// Mitsubishi GX Works2 project: 1111   PLC: Q00J
// 1111111

PROGRAM MAIN
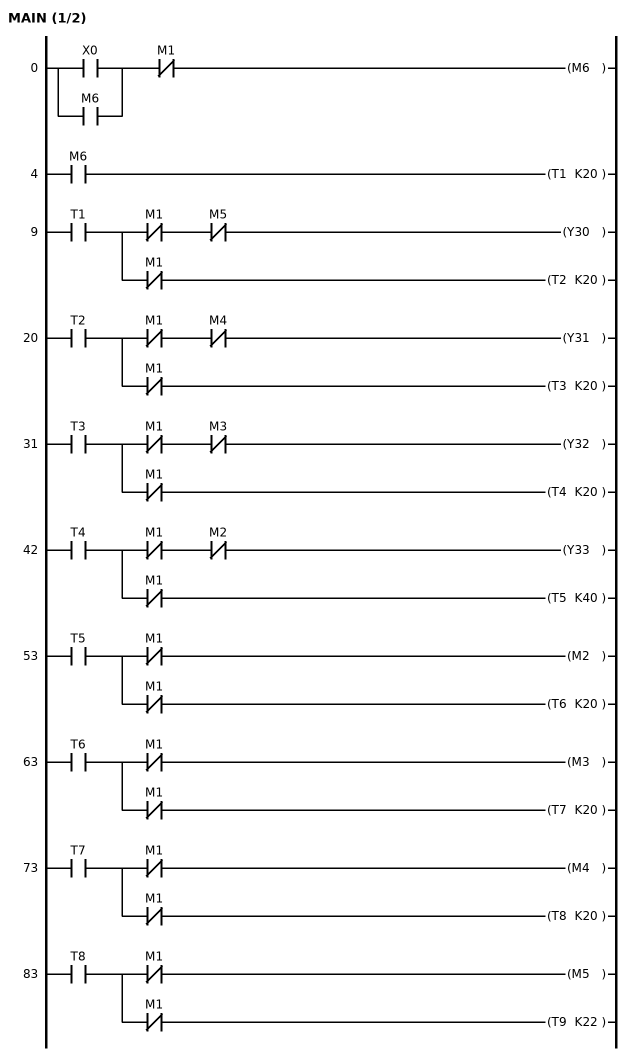
0     LD      X0
      OR      M6
      ANI     M1
      OUT     M6
4     LD      M6
      OUT     T1 K20
9     LD      T1
      MPS
      ANI     M1
      ANI     M5
      OUT     Y30
      MPP
      ANI     M1
      OUT     T2 K20
20    LD      T2
      MPS
      ANI     M1
      ANI     M4
      OUT     Y31
      MPP
      ANI     M1
      OUT     T3 K20
31    LD      T3
      MPS
      ANI     M1
      ANI     M3
      OUT     Y32
      MPP
      ANI     M1
      OUT     T4 K20
42    LD      T4
      MPS
      ANI     M1
      ANI     M2
      OUT     Y33
      MPP
      ANI     M1
      OUT     T5 K40
53    LD      T5
      MPS
      ANI     M1
      OUT     M2
      MPP
      ANI     M1
      OUT     T6 K20
63    LD      T6
      MPS
      ANI     M1
      OUT     M3
      MPP
      ANI     M1
      OUT     T7 K20
73    LD      T7
      MPS
      ANI     M1
      OUT     M4
      MPP
      ANI     M1
      OUT     T8 K20
83    LD      T8
      MPS
      ANI     M1
      OUT     M5
      MPP
      ANI     M1
      OUT     T9 K22
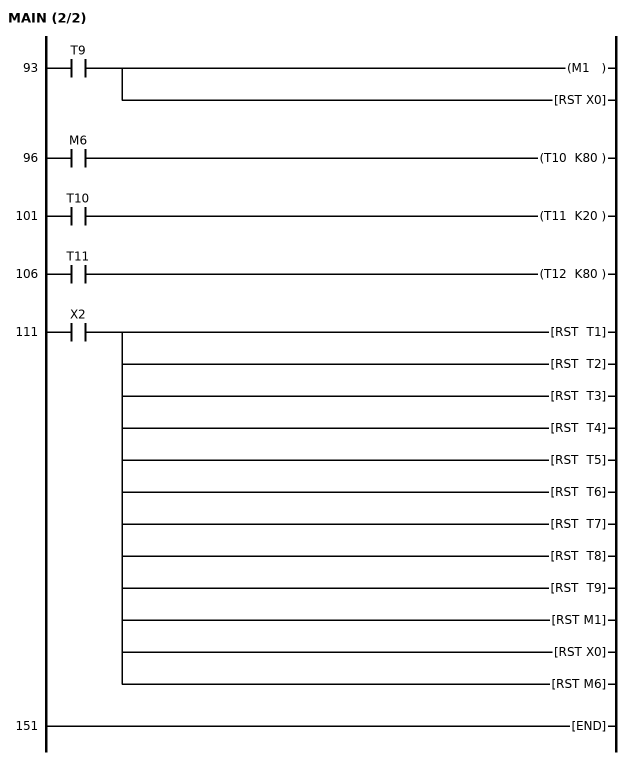
93    LD      T9
      OUT     M1
      RST     X0
96    LD      M6
      OUT     T10 K80
101   LD      T10
      OUT     T11 K20
106   LD      T11
      OUT     T12 K80
111   LD      X2
      RST     T1
      RST     T2
      RST     T3
      RST     T4
      RST     T5
      RST     T6
      RST     T7
      RST     T8
      RST     T9
      RST     M1
      RST     X0
      RST     M6
151   END
END_PROGRAM
